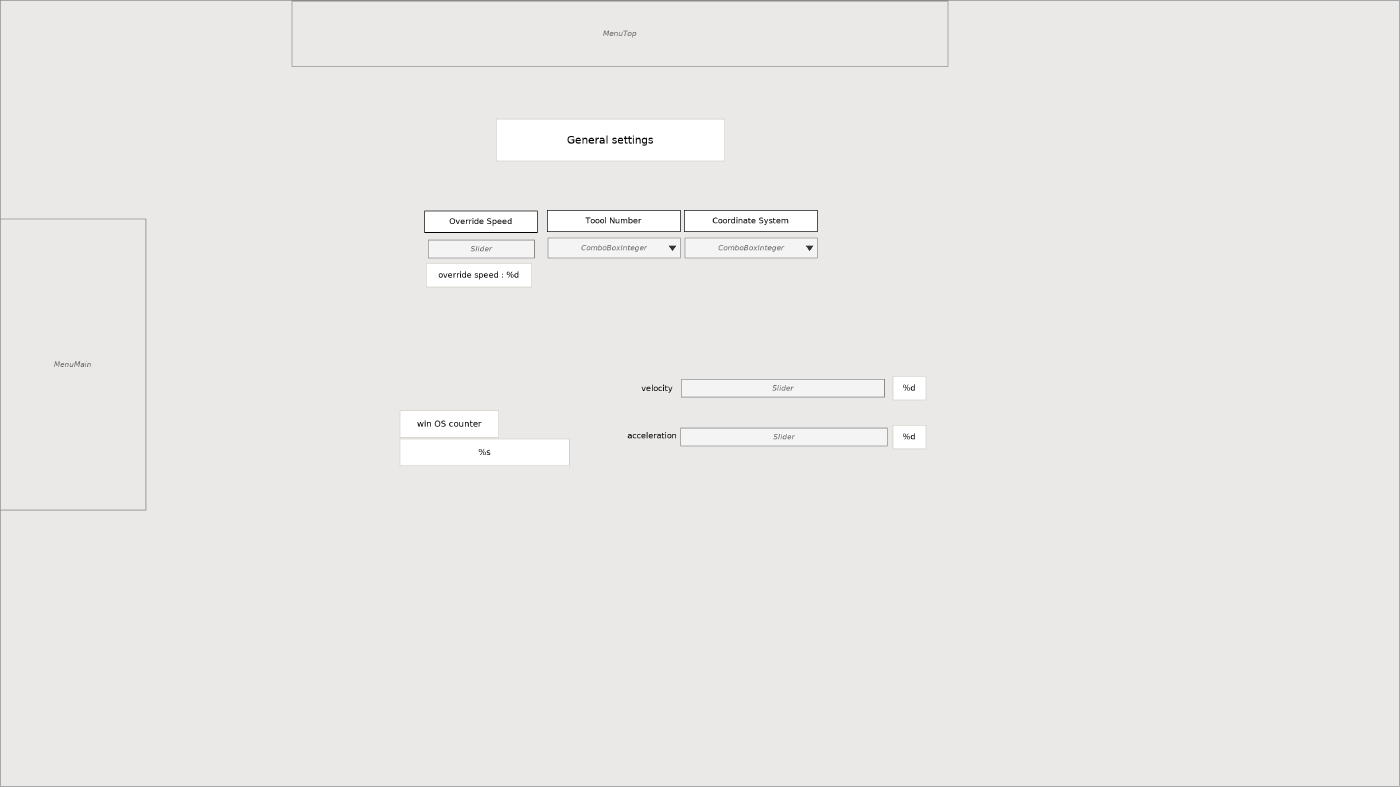
VISUALIZATION APP_Settings  // 1920x1080
    Frame (400,1 900x90)
        shows MenuTop()
    Frame (0,300 200x400)
        shows MenuMain()
    Textfield (680,163 314x58), "General settings"
    Rectangle (582,289 155x30), "Override Speed"
    Rectangle (750,288 183x30), "Toool Number"
    ComboBoxInteger (751,326 182x28), variable: GVL_settings.App_CoordSys.TOOL, text list: 'ToolNumber'
    Slider (934,520 279x25), variable: GVL_settings.App_Velocity, scale 10..50
    Slider (933,587 284x25), variable: GVL_settings.App_Acceleration, scale 10..50
    Label (865,519 72x28), "velocity"
    Label (849,584 91x28), "acceleration"
    Textfield (1224,516 46x33), "%d", text variable: GVL_settings.App_Velocity
    Textfield (1224,583 46x33), "%d", text variable: GVL_settings.App_Acceleration
    Textfield (548,563 136x37), "win OS counter"
    Textfield (548,602 233x37), "%s", text variable: GVL_PLC.Str_windowsCounter
    Rectangle (938,288 183x30), "Coordinate System"
    ComboBoxInteger (939,326 182x28), variable: GVL_settings.App_CoordSys.BASE, text list: 'CoorSys'
    Slider (587,329 146x25), variable: GVL.nOverrideGlobal, scale 10..50
    Textfield (584,361 145x33), "override speed : %d", text variable: GVL.nOverrideGlobal
END_VISUALIZATION

(* stored: Version 1.1.0.1, ProductVersion 3.1.4024.10
   Visu APP_Settings: Id {f7ae8b79-e9cf-4515-af73-0bc3be70ced8} *)
